				END_CASE
			MS_Running :
				IF (NOT sCurrentState.bWaitStep) THEN
(*----------------- Probing ------------------*)
					FOR iSide := 0 TO 1 DO
						CASE aeProbingStep[iSide] OF
							SP_RunStp1 :
								IF abDoProbing[iSide] THEN
									aiProbingCount[iSide] := 0;
									alrProbingStartPos[iSide] := alrTargetPos[PA_Z1 + iSide];
									abProbingDone[iSide] := FALSE;
									abStartPearlingMotor[iSide] := FALSE;
									aeProbingStep[iSide] := SP_RunStp20;
								END_IF
							SP_RunStp20:
								(* Continuous move probing with analog sensor *)
								IF (aTRobotAxis[PA_Z1+ iSide].eCurrentState = AS_InPosition) AND aTWaitMotorStopped[iSide].Q THEN
									(* Move 0.5 mm above probing pos to check default sensor value *)
									alrTargetPos[PA_Z1 + iSide] := alrProbingStartPos[iSide] - 0.5;		// TODO : HFO modifier valeur en dure, original 0.5
									alrCurrentSpeed[PA_Z1 + iSide] := alrMaxRobotSpeed[PA_Z1 + iSide];
									aeMoveRobotCommand[PA_Z1 + iSide] := AC_MoveAtAbsPos;
									aTStickContactValidated[iSide](IN := FALSE);
									aeProbingStep[iSide] := SP_RunStp21;
								END_IF
							SP_RunStp21:
								IF (aTRobotAxis[PA_Z1 + iSide].eCurrentState = AS_InPosition) THEN
									aTStickContactValidated[iSide](IN := TRUE,PT := TStickStabilisationTime);	// Valueur original ==> PT := TStickContactValidTime
									IF aTStickContactValidated[iSide].Q THEN
										asProbingLog[iSide].iPreviousProbingThreshold := aiContactThresholdArea[iSide , aeProbingArea[iSide]];
										aiContactThresholdArea[iSide , aeProbingArea[iSide]] := aiContactDistance[iSide];
										(* Move down 0.5mm *)
										alrTargetPos[PA_Z1 + iSide] := alrProbingStartPos[iSide]- 0.3;  		// TODO : HFO, Ajout de valeur negative
										//alrTargetPos[PA_Z1 + iSide] := alrProbingStartPos[iSide];
										aeMoveRobotCommand[PA_Z1 + iSide] := AC_MoveAtAbsPos;
										aTStickContactValidated[iSide](IN := FALSE);
										aeProbingStep[iSide] := SP_RunStp25;
									END_IF
								END_IF
							SP_RunStp25:
								IF (aTRobotAxis[PA_Z1 + iSide].eCurrentState = AS_InPosition) THEN
									aTStickContactValidated[iSide](IN := TRUE,PT := TStickContactValidTime);
									IF aTStickContactValidated[iSide].Q THEN
										(* Check if we must go up or down *)
										IF (aiContactDistance[iSide] > aiContactThresholdArea[iSide , aeProbingArea[iSide]] + alrSensorRate[iSide] * lrProbingThreshold) THEN
											(* Go up *)
											aeProbingStep[iSide] := SP_RunStp30;
										ELSE
											(* Go down *)
											aeProbingStep[iSide] := SP_RunStp40;
										END_IF								
									END_IF
								END_IF	
							SP_RunStp30:
								(* Move up slowly until we get contact *)
								alrTargetPos[PA_Z1 + iSide] := alrProbingStartPos[iSide] - 2;
								alrCurrentSpeed[PA_Z1 + iSide] := lrSensorZSpeed;
								aeMoveRobotCommand[PA_Z1 + iSide] := AC_MoveAtAbsPos;
								aeProbingStep[iSide] := SP_RunStp35;
							SP_RunStp35:
								IF (aiContactDistance[iSide] < aiContactThresholdArea[iSide , aeProbingArea[iSide]] + alrSensorRate[iSide] * lrProbingThreshold) THEN
									aTStickContactValidated[iSide](IN := FALSE);
									aeMoveRobotCommand[PA_Z1 + iSide] := AC_Stop;
									aeProbingStep[iSide] := SP_RunStp50;
									sCurrentState.bWaitStep := TRUE;
								ELSIF (aTRobotAxis[PA_Z1 + iSide].eCurrentState = AS_InPosition) THEN
									aeMoveRobotCommand[PA_Z1] := AC_Stop;
									aeMoveRobotCommand[PA_Z2] := AC_Stop;
									bSecurityError := TRUE;
									iDebugPos := 1;
									iDebugSide := iSide;
								END_IF
							SP_RunStp40:
								(* Move down slowly until we get contact *)
								alrTargetPos[PA_Z1 + iSide] := alrProbingLimit[iSide];
								alrCurrentSpeed[PA_Z1 + iSide] := lrSensorZSpeed;
								aeMoveRobotCommand[PA_Z1 + iSide] := AC_MoveAtAbsPos;
								aeProbingStep[iSide] := SP_RunStp45;
							SP_RunStp45:
								IF (aiContactDistance[iSide] > aiContactThresholdArea[iSide , aeProbingArea[iSide]] + alrSensorRate[iSide] * lrProbingThreshold) THEN
									aTStickContactValidated[iSide](IN := FALSE);
									aeMoveRobotCommand[PA_Z1 + iSide] := AC_Stop;
									aeProbingStep[iSide] := SP_RunStp50;
									sCurrentState.bWaitStep := TRUE;
								ELSIF (aTRobotAxis[PA_Z1 + iSide].eCurrentState = AS_InPosition) THEN
									aeMoveRobotCommand[PA_Z1] := AC_Stop;
									aeMoveRobotCommand[PA_Z2] := AC_Stop;
									bSecurityError := TRUE;
									iDebugPos := 10;
									iDebugSide := iSide;
								END_IF
							SP_RunStp50:
								IF (aTRobotAxis[PA_Z1 + iSide].eCurrentState = AS_InPosition) THEN
									aTStickContactValidated[iSide](IN := TRUE,PT := TStickContactValidTime);
									IF aTStickContactValidated[iSide].Q THEN
										alrProbingPos[iSide] := aTRobotAxis[PA_Z1 + iSide].lrCurrentPos - (aiContactDistance[iSide] - aiContactThresholdArea[iSide , aeProbingArea[iSide]])/alrSensorRate[iSide];
										(* Move 2 mm above probing pos to check 1st measure *)
										alrTargetPos[PA_Z1 + iSide] := aTRobotAxis[PA_Z1 + iSide].lrCurrentPos - 2;
										alrCurrentSpeed[PA_Z1 + iSide] := alrMaxRobotSpeed[PA_Z1 + iSide];
										aeMoveRobotCommand[PA_Z1 + iSide] := AC_MoveAtAbsPos;
										aeProbingStep[iSide] := SP_RunStp55;
									END_IF
								END_IF
							SP_RunStp55:
								IF (aTRobotAxis[PA_Z1 + iSide].eCurrentState = AS_InPosition) AND NOT asProbingLog[iSide].bNewLog THEN
									(* Move to contact position *)
									alrTargetPos[PA_Z1 + iSide] := alrTargetPos[PA_Z1 + iSide]+2;
									aeMoveRobotCommand[PA_Z1 + iSide] := AC_MoveAtAbsPos;
									aTStickContactValidated[iSide](IN := FALSE);
									aeProbingStep[iSide] := SP_RunStp60;
								END_IF
							SP_RunStp60:
								IF (aTRobotAxis[PA_Z1 + iSide].eCurrentState = AS_InPosition) THEN
									aTStickContactValidated[iSide](IN := TRUE,PT := TStickContactValidTime);
									IF aTStickContactValidated[iSide].Q THEN
										alrCheckProbingPos[iSide] := aTRobotAxis[PA_Z1 + iSide].lrCurrentPos - (aiContactDistance[iSide] - aiContactThresholdArea[iSide , aeProbingArea[iSide]])/alrSensorRate[iSide];
										asProbingLog[iSide].alrProbingPos[PH_Left] := alrProbingPos[iSide];
										asProbingLog[iSide].alrProbingPos[PH_Right] := alrCheckProbingPos[iSide];
										asProbingLog[iSide].eProbingArea := aeProbingArea[iSide];
										asProbingLog[iSide].iProbingThreshold := aiContactThresholdArea[iSide , aeProbingArea[iSide]];
										asProbingLog[iSide].bNewLog := TRUE;
(* DLA										IF (ABS(alrProbingPos[iSide] - alrCheckProbingPos[iSide]) < 0.1) THEN *)
										IF (ABS(alrProbingPos[iSide] - alrCheckProbingPos[iSide]) < 0.3) THEN
											abProbingDone[iSide] := TRUE;
											aeProbingStep[iSide] := SP_RunStp70;
										ELSIF abRetryProbing[iSide] AND aiProbingCount[iSide] < 3 AND (ABS(alrProbingPos[iSide] - alrCheckProbingPos[iSide]) < 0.3)THEN
											aiProbingCount[iSide] := aiProbingCount[iSide] + 1;
											aeProbingStep[iSide] := SP_RunStp20;
										ELSE
											bSecurityError := TRUE;
											iDebugPos := 2;
											iDebugSide := iSide;
										END_IF
									END_IF
								END_IF
							SP_RunStp70:
								IF NOT abDoProbing[iSide] THEN
									aeProbingStep[iSide] := SP_RunStp1;
								END_IF
						END_CASE
					END_FOR
(*----------------- Stick gestion ------------------*)
					CASE eStickStep OF
						SP_RunStp1 :
							IF (aTRobotAxis[PA_Z1].eCurrentState = AS_InPosition) AND (aTRobotAxis[PA_Z2].eCurrentState = AS_InPosition) THEN
								FOR iSide := 0 TO 1 DO
									IF abChangeStick[iSide] AND abUseSpindle[iSide] THEN
										abSharpenStick[iSide] := TRUE;
										eStickStep := SP_RunStp2; (* Change Stick [Serial]*)
									END_IF
								END_FOR
								IF (eStickStep <> SP_RunStp2) THEN
									FOR iSide := 0 TO 1 DO
										IF abSharpenStick[iSide] AND abUseSpindle[iSide] THEN
											IF NOT abChuckClosed[iSide] THEN
												abSharpenStick[iSide] := FALSE;
											ELSE
												IF abNewStick[iSide] OR aiNbOfPearlsDone[iSide]>0 THEN
													eStickStep := SP_RunStp50; (* Sharpen [parallel]*)
												ELSIF NOT abNewStick[iSide] AND abSharpenStick[iSide] AND aiNbOfPearlsDone[iSide]=0 THEN
													(* sharpen is not need if no pearl has been made *)
													abSharpenStick[iSide] := FALSE;
												END_IF
											END_IF
										END_IF
									END_FOR
								END_IF
							END_IF
						SP_RunStp2 : (* Change Stick [Serial]*)
							FOR iSide := 0 TO 1 DO
								(* Stop motors *)
								abStartPearlingMotor[iSide] := FALSE;
								(* Move Z to safe *)
								alrTargetPos[PA_Z1+iSide] := alrSafePos[PA_Z1+iSide];
								aeMoveRobotCommand[PA_Z1+iSide] := AC_MoveAtAbsPos;
							END_FOR
							eStickStep := SP_RunStp10;
						SP_RunStp10 :  (* Reject Stick [Serial]*)
							IF (aTRobotAxis[PA_Z1].eCurrentState = AS_InPosition) AND
									(aTRobotAxis[PA_Z2].eCurrentState = AS_InPosition) THEN
								eStickStep := SP_RunStp20; (* Nothing to reject, Get new Stick *)
								FOR iSide := 0 TO 1 DO
									(* First drop stick if any *)
									IF abChuckClosed[iSide] AND abChangeStick[iSide] AND abUseSpindle[iSide] THEN
										iRejectPos := iSide;
										eStickStep := SP_RunStp11; (* First drop stick if any *)
										EXIT;
									END_IF
								END_FOR
							END_IF
						SP_RunStp11 :
							(* Move to reject *)
							alrTargetPos[PA_X] := alrRobotPos[PA_X,PTP_RejectPosZ1+iRejectPos];
							alrTargetPos[PA_Y] := alrRobotPos[PA_Y,PTP_RejectPosZ1+iRejectPos];
							aeMoveRobotCommand[PA_X] := AC_MoveAtAbsPos;
							aeMoveRobotCommand[PA_Y] := AC_MoveAtAbsPos;
							eStickStep := SP_RunStp12;
						SP_RunStp12 :
							IF (eRobotXYStatus = AS_InPosition) THEN
								(* Move Z to reject pos *)
								alrTargetPos[PA_Z1+iRejectPos] := alrRobotPos[PA_Z1 + iRejectPos,PTP_RejectPosZ1+iRejectPos];
								aeMoveRobotCommand[PA_Z1+iRejectPos] := AC_MoveAtAbsPos;
								eStickStep := SP_RunStp13;
							END_IF
						SP_RunStp13 :
							IF (aTRobotAxis[PA_Z1+iRejectPos].eCurrentState = AS_InPosition) THEN
								(* Open chuck *)
								abOpenChuck[iRejectPos] := TRUE;
								TCheckTimer(IN := FALSE);
								eStickStep := SP_RunStp14;
							END_IF
						SP_RunStp14 :
							IF abChuckOpened[iRejectPos] THEN
								abActivateEject[iRejectPos] := TRUE;
								TCheckTimer(IN := TRUE,PT := TCheckTime);
								IF TCheckTimer.Q THEN
									abActivateEject[iRejectPos] := FALSE;
									alrTargetPos[PA_Z1+iRejectPos] := alrSafePos[PA_Z1+iRejectPos];
									aeMoveRobotCommand[PA_Z1+iRejectPos] := AC_MoveAtAbsPos;
									eStickStep :=  SP_RunStp10;
								END_IF
							ELSE
								TCheckTimer(IN := FALSE);
							END_IF
						SP_RunStp20 :  (* Get new stick [Serial]*)
							IF (aTRobotAxis[PA_Z1].eCurrentState = AS_InPosition) AND
									(aTRobotAxis[PA_Z2].eCurrentState = AS_InPosition) THEN
								eStickStep := SP_RunStp1; (* Nothing to change *)
								FOR iSide := 0 TO 1 DO
									IF abChangeStick[iSide]  AND abUseSpindle[iSide] THEN
										iChangeStickPos := iSide;
										eStickStep := SP_RunStp21; (* Get new stick *)
										EXIT;
									END_IF
								END_FOR
							END_IF
						SP_RunStp21 :
							iStickHead := iChangeStickPos+1;
							eBarrelRunCmd := RCB_PrepareStick;
							alrTargetPos[PA_X] := alrRobotPos[PA_X,PTP_BarrelPosZ1+iChangeStickPos];
							alrTargetPos[PA_Y] := alrRobotPos[PA_Y,PTP_BarrelPosZ1+iChangeStickPos];
							aeMoveRobotCommand[PA_X] := AC_MoveAtAbsPos;
							aeMoveRobotCommand[PA_Y] := AC_MoveAtAbsPos;
							eStickStep := SP_RunStp22;
						SP_RunStp22 :
							IF (eRobotXYStatus = AS_InPosition) AND (eBarrelRunStatus= RS_WaitRequest ) THEN
								sOutTakeFromBarrel.bHasTaken := FALSE;
								sOutTakeFromBarrel.bReadyToTake := FALSE;
								eBarrelRunCmd := RCB_GiveStick;
								eStickStep := SP_RunStp23;
							END_IF
						SP_RunStp23 :
							IF (eRobotXYStatus = AS_InPosition)  THEN
								(* Move Z to stick pos *)
								alrTargetPos[PA_Z1+iChangeStickPos] := alrRobotPos[PA_Z1+iChangeStickPos,PTP_BarrelPosZ1+iChangeStickPos];
								aeMoveRobotCommand[PA_Z1+iChangeStickPos] := AC_MoveAtAbsPos;
								eStickStep := SP_RunStp24;
							END_IF
						SP_RunStp24 :
							IF (ABS(aTRobotAxis[PA_Z1+iChangeStickPos].lrCurrentPos - alrTargetPos[PA_Z1+iChangeStickPos]) <= 10) THEN
								(* reduce speed when take stick *)
								alrCurrentSpeed[PA_Z1+iChangeStickPos] := lrStickTakeSpeed;
							END_IF
							IF (aTRobotAxis[PA_Z1+iChangeStickPos].eCurrentState = AS_InPosition) THEN
								alrCurrentSpeed := alrMaxRobotSpeed;
								sOutTakeFromBarrel.bReadyToTake := TRUE;
								eStickStep := SP_RunStp25;
							END_IF
						SP_RunStp25 :
							IF sInTakeFromBarrel.bHasGiven THEN
								(* Close chuck *)
								abOpenChuck[iChangeStickPos] := FALSE;
								eStickStep := SP_RunStp26;
							END_IF
						SP_RunStp26 :
							IF abChuckClosed[iChangeStickPos] THEN
								abNewStick[iChangeStickPos] := TRUE;
								(* Move Z to safe *)
								alrTargetPos[PA_Z1+iChangeStickPos] := alrSafePos[PA_Z1+iChangeStickPos];
								aeMoveRobotCommand[PA_Z1+iChangeStickPos] := AC_MoveAtAbsPos;
								eStickStep := SP_RunStp27;
							END_IF
						SP_RunStp27 :
							IF (aTRobotAxis[PA_Z1+iChangeStickPos].eCurrentState = AS_InPosition) THEN
								sOutTakeFromBarrel.bHasTaken := TRUE;
								eStickStep := SP_RunStp28;
							END_IF
						SP_RunStp28 :
							IF eBarrelRunStatus = RS_WaitRequest  THEN
								IF sInTakeFromBarrel.bHasGiven THEN
									abChangeStick[iChangeStickPos] := FALSE;
									abSharpenStick[iChangeStickPos] := TRUE;
									alrRemainingStickLength[iChangeStickPos] := asStickData[iChangeStickPos].lrTotalLength;
									eStickStep := SP_RunStp20;
								ELSE
									bStickNotTakenError := TRUE;
									abSpindleError[iChangeStickPos] := TRUE;
									abOpenChuck[iChangeStickPos] := TRUE;
									eStickStep := SP_RunStp1;  (*Error *)
								END_IF
							END_IF
						SP_RunStp50 : (* Sharpen [parallel]*)
							IF (eSharpenRunStatus =  RS_WaitRequest) THEN
								FOR iSide := 0 TO 1 DO
									(* Stop motors *)
									abStartPearlingMotor[iSide] := FALSE;
									(* Move Z to safe *)
									alrTargetPos[PA_Z1+iSide] := alrSafePos[PA_Z1+iSide];
									aeMoveRobotCommand[PA_Z1+iSide] := AC_MoveAtAbsPos;
								END_FOR
								eStickStep := SP_RunStp51;
							END_IF
						SP_RunStp51 :
							IF (aTRobotAxis[PA_Z1].eCurrentState = AS_InPosition) AND
									(aTRobotAxis[PA_Z2].eCurrentState = AS_InPosition) THEN
								alrTargetPos[PA_X] := alrRobotPos[PA_X,PTP_Sharpen];
								alrTargetPos[PA_Y] := alrRobotPos[PA_Y,PTP_Sharpen];
								aeMoveRobotCommand[PA_X] := AC_MoveAtAbsPos;
								aeMoveRobotCommand[PA_Y] := AC_MoveAtAbsPos;
								eStickStep := SP_RunStp52;
							END_IF
						SP_RunStp52 :
							IF (eRobotXYStatus = AS_InPosition)  THEN
								(* Move Z to sharpen pos if needed*)
								FOR iSide := 0 TO 1 DO
									IF abSharpenStick[iSide]  AND abUseSpindle[iSide] THEN
										(* After sharpening, pearling correction must be recalculated *)
										alrCorrectionMCR[iSide] := 0;
										IF abNewStick[iSide] THEN
											alrTargetPos[PA_Z1+iSide] := alrRobotPos[PA_Z1+iSide,PTP_Sharpen] - lrStickOutAfterChange - 0.5;
										ELSE
											alrTargetPos[PA_Z1+iSide] := alrRobotPos[PA_Z1+iSide,PTP_Sharpen] - lrSharpenPosOffset - asStickData[iSide].lrOutLength;
										END_IF
										aeMoveRobotCommand[PA_Z1+iSide] := AC_MoveAtAbsPos;
									END_IF
								END_FOR
								alrCurrentSpeed := alrMaxRobotSpeed;
								eStickStep := SP_RunStp53;
							END_IF
						SP_RunStp53 :
							IF (aTRobotAxis[PA_Z1].eCurrentState = AS_InPosition) AND
									(aTRobotAxis[PA_Z2].eCurrentState = AS_InPosition) THEN
								FOR iSide := 0 TO 1 DO
									IF abSharpenStick[iSide]  AND abUseSpindle[iSide] THEN
										IF NOT abNewStick[iSide] THEN
											alrProbingLimit[iSide] :=  alrRobotPos[PA_Z1+iSide,PTP_Sharpen] + 0.5;
											abDoProbing[iSide] := TRUE;
											abRetryProbing[iSide] := FALSE;
										END_IF
										aeProbingArea[iSide] := PA_BeforeSharpen;
									END_IF
								END_FOR
								eStickStep := SP_RunStp54;
							END_IF
						SP_RunStp54 :
							IF (abProbingDone[PH_Left] OR NOT abSharpenStick[PH_Left] OR NOT abUseSpindle[PH_Left] OR abNewStick[PH_Left]) AND (abProbingDone[PH_Right] OR NOT abSharpenStick[PH_Right] OR  NOT abUseSpindle[PH_Right] OR abNewStick[PH_Right]) THEN
								FOR iSide := 0 TO 1 DO
									abDoProbing[iSide] := FALSE;
									(* We have the right position, calculate stick use *)
									IF abSharpenStick[iSide]   AND abUseSpindle[iSide] THEN
										IF abNewStick[iSide] THEN
											alrRemainingStickLength[iSide] := asStickData[iSide].lrTotalLength;
										ELSE
											IF (alrProbingPos[iSide] - alrLastProbingPos[iSide]) > (asStickData[iSide].lrOutLength -0.5) THEN
												alrRemainingStickLength[iSide] := sStickDataShared.sStickDataMMIShared.lrMinHoldLength;
											ELSE
												alrRemainingStickLength[iSide] := alrRemainingStickLength[iSide] - (alrProbingPos[iSide] - alrLastProbingPos[iSide]);
											END_IF
										END_IF
										(* Check if it is the first probing after stick change *)
										IF (alrRemainingStickLength[iSide] > asStickData[iSide].lrTotalLength) THEN
											alrRemainingStickLength[iSide] := asStickData[iSide].lrTotalLength;
										END_IF
										(* Check if the stick is not too short *)
										IF (alrRemainingStickLength[iSide] < (sStickDataShared.sStickDataMMIShared.lrMinHoldLength + asStickData[iSide].lrOutLength)) THEN
											(* We must change the stick *)
											abChangeStick[iSide] := TRUE;
											abSharpenStick[iSide] := FALSE;
											eStickStep := SP_RunStp1;
										END_IF
									END_IF
								END_FOR
								IF (eStickStep = SP_RunStp1) THEN
									(* In parallel pearling, we must change both stick *)
									IF bParallelProduction THEN
										FOR iSide:=0 TO 1 DO
											abChangeStick[iSide] := TRUE;
											abSharpenStick[iSide] := FALSE;
										END_FOR
									END_IF
								ELSE
									FOR iSide := 0 TO 1 DO
										IF abSharpenStick[iSide]   AND abUseSpindle[iSide] AND NOT abNewStick[iSide] THEN
											alrTargetPos[PA_Z1+iSide] := alrTargetPos[PA_Z1+iSide] - 0.5;
											aeMoveRobotCommand[PA_Z1+iSide] := AC_MoveAtAbsPos;
										END_IF
									END_FOR
									eStickStep := SP_RunStp55;
								END_IF
							END_IF
						SP_RunStp55 :
							IF (aTRobotAxis[PA_Z1].eCurrentState = AS_InPosition) AND
								(aTRobotAxis[PA_Z2].eCurrentState = AS_InPosition) THEN
								FOR iSide := 0 TO 1 DO
									IF   abUseSpindle[iSide] AND abSharpenStick[iSide] THEN
										(* Open chuck *)
										abOpenChuck[iSide] := TRUE;
									END_IF
								END_FOR
								TWaitChuckOpen(IN := FALSE);
								eStickStep := SP_RunStp56;
							END_IF
						SP_RunStp56 :
							TWaitChuckOpen(IN := (abChuckOpened[PH_Left] OR NOT abOpenChuck[PH_Left] OR NOT abUseSpindle[PH_Left]) AND (abChuckOpened[PH_Right] OR NOT abOpenChuck[PH_Right] OR NOT abUseSpindle[PH_Right]),PT := T#400MS);   // Valeur de départ ==> PT := t#1s
							FOR iSide := 0 TO 1 DO
								IF abUseSpindle[iSide] AND abSharpenStick[iSide] THEN
									abActivateEject[iSide] := abChuckOpened[iSide] AND abOpenChuck[iSide];
									IF  TWaitChuckOpen.Q THEN
										(* Move Z to out position *)
										alrCurrentSpeed := alrMaxRobotSpeed;
										alrTargetPos[PA_Z1+iSide] := alrRobotPos[PA_Z1+iSide,PTP_Sharpen]- asStickData[iSide].lrOutLength - alrSharpenTeachZOffset;
										aeMoveRobotCommand[PA_Z1+iSide] := AC_MoveAtAbsPos;
										//eStickStep := SP_RunStp57;		// HFO : Supprimer la correction avec capteur step 57, 58, 24.11.2021
										eStickStep := SP_RunStp59;
									END_IF
								END_IF
							END_FOR
						SP_RunStp57:
							IF (aTRobotAxis[PA_Z1].eCurrentState = AS_InPosition) AND
								(aTRobotAxis[PA_Z2].eCurrentState = AS_InPosition) THEN
								TWaitHeadStab(IN := FALSE);
								eStickStep := SP_RunStp58;
							END_IF
						SP_RunStp58:
							TWaitHeadStab(IN := TRUE, PT := T#150MS);	// Valeur de départ ==> PT := t#500ms
							IF TWaitHeadStab.Q THEN
								FOR iSide := 0 TO 1 DO
									IF abUseSpindle[iSide] AND abSharpenStick[iSide] THEN
										alrTargetPos[PA_Z1+iSide] := alrTargetPos[PA_Z1+iSide] + (aiContactDistance[iSide] - aiContactThresholdArea[iSide , aeProbingArea[iSide]])/alrSensorRate[iSide] - alrChuckRetractOffset[iSide];
										aeMoveRobotCommand[PA_Z1+iSide] := AC_MoveAtAbsPos;
									END_IF
								END_FOR
								eStickStep := SP_RunStp59;
							END_IF
						SP_RunStp59:
							IF (aTRobotAxis[PA_Z1].eCurrentState = AS_InPosition) AND
									(aTRobotAxis[PA_Z2].eCurrentState = AS_InPosition) THEN
								TWaitHeadStab(IN := FALSE);
								eStickStep := SP_RunStp60;
							END_IF
						SP_RunStp60:
							TWaitHeadStab(IN := TRUE, PT := T#400MS);	// Valeur de départ ==> PT := t#500ms
							IF TWaitHeadStab.Q THEN
								eStickStep := SP_RunStp61;
							END_IF
						SP_RunStp61 :
							IF (aTRobotAxis[PA_Z1].eCurrentState = AS_InPosition) AND
									(aTRobotAxis[PA_Z2].eCurrentState = AS_InPosition) THEN
								(* Close chuck if needed*)
								FOR iSide := 0 TO 1 DO
									IF abUseSpindle[iSide] AND abSharpenStick[iSide] THEN
										abOpenChuck[iSide] := FALSE;
									END_IF
								END_FOR
								IF (abChuckClosed[PH_Left]  OR abOpenChuck[PH_Left] OR NOT abUseSpindle[PH_Left]) AND (abChuckClosed[PH_Right] OR abOpenChuck[PH_Right] OR NOT abUseSpindle[PH_Right]) THEN
									FOR iSide := 0 TO 1 DO
										IF abUseSpindle[iSide] AND abSharpenStick[iSide] THEN
											(* Retract ejector *)
											abActivateEject[iSide] := FALSE;
											(* Do probing *)
											alrTargetPos[PA_Z1+iSide] := alrTargetPos[PA_Z1+iSide];
(* DLA : Remove -1mm for optimisation 											alrTargetPos[PA_Z1+iSide] := alrTargetPos[PA_Z1+iSide] - 1;*)
											alrProbingLimit[iSide] :=  alrRobotPos[PA_Z1+iSide,PTP_Sharpen] - 0.5;
											abDoProbing[iSide] := TRUE;
											abRetryProbing[iSide] := FALSE;
											aeProbingArea[iSide] := PA_AfterSharpen;
										END_IF
									END_FOR
									eStickStep := SP_RunStp62;
								END_IF
							END_IF
						SP_RunStp62 :
							IF (abProbingDone[PH_Left] OR NOT abSharpenStick[PH_Left]  OR NOT abUseSpindle[PH_Left]) AND (abProbingDone[PH_Right] OR NOT abSharpenStick[PH_Right] OR NOT abUseSpindle[PH_Right]) THEN
								alrCurrentSpeed := alrMaxRobotSpeed;
								FOR iSide := 0 TO 1 DO
									IF abUseSpindle[iSide] AND abSharpenStick[iSide] THEN
										alrLastProbingPos[iSide] := alrProbingPos[iSide];
										alrSharpenProbing[iSide] := alrProbingPos[iSide];
										alrStickCorrection[iSide] := alrRobotPos[PA_Z1+iSide,PTP_Sharpen]  - alrProbingPos[iSide] - asStickData[iSide].lrOutLength - alrSharpenTeachZOffset;
										(* Move down to sharpen end position*)
										alrTargetPos[PA_Z1+iSide] := alrProbingPos[iSide] - 0.1;
										aeMoveRobotCommand[PA_Z1+iSide] := AC_MoveAtAbsPos;
										(* Check if there is a risk for the spindle or stick is stuck in the chuck*)
										IF (alrProbingPos[iSide] > ( alrRobotPos[PA_Z1+iSide,PTP_Sharpen] - (asStickData[iSide].lrOutLength - 0.5))) THEN
											abChangeStick[iSide] := TRUE;
											bSecurityError := TRUE;
											iDebugPos := 3;
											iDebugSide := iSide;
										END_IF
									END_IF
								END_FOR
								IF bSecurityError THEN
									aeMoveRobotCommand[PA_Z1] := AC_None;
									aeMoveRobotCommand[PA_Z2] := AC_None;
								ELSE
									bAspirationSharpenOn := TRUE;
									eStickStep := SP_RunStp63;
								END_IF
							END_IF
						SP_RunStp63 :
							IF (aTRobotAxis[PA_Z1].eCurrentState = AS_InPosition) AND
									(aTRobotAxis[PA_Z2].eCurrentState = AS_InPosition) THEN
								IF bUseFullTapeWidth THEN
									(* Move to start position *)
									alrCurrentSpeed := alrMaxRobotSpeed;
									alrTargetPos[PA_Y] := alrRobotPos[PA_Y,PTP_Sharpen] - lrCenterSharpningOffset - lrSharpeningDelta;
									aeMoveRobotCommand[PA_Y] := AC_MoveAtAbsPos;
								END_IF
								yMCRChannel := 1;
								eStickStep := SP_RunStp64;
							END_IF
						SP_RunStp64 :
							eMCRCommand := MCRC_SetSpeed;
							TMCRDrv.iSpeedSetpoint :=  sStickDataShared.sStickDataMMIShared.iMCRSharpenSpeed;
							eStickStep := SP_RunStp65;
						SP_RunStp65 :
							IF bMCRReady THEN
								IF yMCRChannel = 1 THEN
									yMCRChannel := 2;
									eStickStep := SP_RunStp64;
								ELSE
									yMCRChannel := 1;
									eStickStep := SP_RunStp66;
								END_IF
							END_IF
						SP_RunStp66:
							(* Wait XY in start position *)
							IF (eRobotXYStatus = AS_InPosition) THEN
								FOR iSide := 0 TO 1 DO
									IF abUseSpindle[iSide] AND abSharpenStick[iSide] THEN
										abStartPearlingMotor[iSide] := TRUE;
									END_IF
								END_FOR
								IF  (aTWaitMotorStarted[PH_Left].Q OR NOT abSharpenStick[PH_Left] OR NOT abUseSpindle[PH_Left]) AND (aTWaitMotorStarted[PH_Right].Q OR NOT abSharpenStick[PH_Right] OR NOT abUseSpindle[PH_Right])   THEN
									FOR iSide := 0 TO 1 DO
										IF abUseSpindle[iSide] AND abSharpenStick[iSide] THEN
											abDoProbing[iSide] := FALSE;
											(* Move down to sharpen end position*)
											IF abNewStick[iSide] THEN
												alrTargetPos[PA_Z1+iSide] := alrTargetPos[PA_Z1+iSide] + 0.2 +0.05;
											ELSE
												alrTargetPos[PA_Z1+iSide] := alrTargetPos[PA_Z1+iSide] + sStickDataShared.sStickDataMMIShared.lrSharpenHeight+0.05;
											END_IF
											aeMoveRobotCommand[PA_Z1+iSide] := AC_MoveAtAbsPos;
											abNewStick[iSide] := FALSE;
										END_IF
									END_FOR
									alrCurrentSpeed := alrMaxRobotSpeed;
									iNbOfFwBwSharpen := 0;
									iNbOfFwBwSharpenBeforeMove := 0;
									eStickStep := SP_RunStp67;
								END_IF
							END_IF
						SP_RunStp67 :
							IF  (aTRobotAxis[PA_Z1].eCurrentState = AS_InPosition) AND (aTRobotAxis[PA_Z2].eCurrentState = AS_InPosition) THEN
								(* Reduce speed for sharpening *)
								alrCurrentSpeed[PA_Y] := sStickDataShared.sStickDataMMIShared.lrSharpenSpeed;
								eStickStep := SP_RunStp68;
							END_IF
						SP_RunStp68 :
							(* Do sharpening *)
							IF (eRobotXYStatus = AS_InPosition) THEN
								iNbOfFwBwSharpen := iNbOfFwBwSharpen+1;
								iNbOfFwBwSharpenBeforeMove := iNbOfFwBwSharpenBeforeMove + 1;
								(* Check if sharpen is finished *)
								IF (iNbOfFwBwSharpen >  sStickDataShared.sStickDataMMIShared.iNbOfFwBwSharpen) THEN
									eStickStep := SP_RunStp71;
								ELSE
									eStickStep := SP_RunStp69;
									IF bUseFullTapeWidth THEN
										IF iNbOfFwBwSharpen = 1 THEN
											alrTargetPos[PA_Y] := alrRobotPos[PA_Y,PTP_Sharpen] - lrCenterSharpningOffset - lrSharpeningDelta;
											eStickStep := SP_RunStp80;
										ELSE
											alrTargetPos[PA_Y] := alrRobotPos[PA_Y,PTP_Sharpen] - lrCenterSharpningOffset;
										END_IF
									ELSE
										alrTargetPos[PA_Y] := alrRobotPos[PA_Y,PTP_Sharpen] - lrCenterSharpningOffset + lrSharpeningDelta;
									END_IF
									aeMoveRobotCommand[PA_Y] := AC_MoveAtAbsPos;
								END_IF
							END_IF
						SP_RunStp69 :
							(* Do sharpening *)
							IF (eRobotXYStatus = AS_InPosition) THEN
								eStickStep := SP_RunStp68;
								IF (iNbOfFwBwSharpenBeforeMove >= sStickDataShared.sStickDataMMIShared.iNbOfFwBwBeforeTapeMove) OR
											(iNbOfFwBwSharpen = sStickDataShared.sStickDataMMIShared.iNbOfFwBwSharpen) THEN
									IF bUseFullTapeWidth THEN
										(* Move on clean tape part *)
										alrTargetPos[PA_Y] := alrRobotPos[PA_Y,PTP_Sharpen] - lrCenterSharpningOffset + lrSharpeningDelta;
										aeMoveRobotCommand[PA_Y] := AC_MoveAtAbsPos;
									ELSE
										(* Move Sharpen Tape*)
										eSharpenRunCmd := RCS_MoveStep;
										eStickStep := SP_RunStp70;
									END_IF
									iNbOfFwBwSharpenBeforeMove := 0;
								ELSIF bUseFullTapeWidth THEN
									(* Move BW *)
									alrTargetPos[PA_Y] := alrRobotPos[PA_Y,PTP_Sharpen] - lrCenterSharpningOffset - lrSharpeningDelta;
									aeMoveRobotCommand[PA_Y] := AC_MoveAtAbsPos;
								END_IF
							END_IF
						SP_RunStp70 :
							IF eSharpenRunStatus =  RS_WaitRequest THEN
								alrTargetPos[PA_Y] := alrRobotPos[PA_Y,PTP_Sharpen];
								aeMoveRobotCommand[PA_Y] := AC_MoveAtAbsPos;
								eStickStep := SP_RunStp68;
							END_IF
						SP_RunStp71 :
							(* End of  sharpening *)
							IF (eRobotXYStatus = AS_InPosition) THEN
								IF bUseFullTapeWidth THEN
									(* Move Sharpen Tape*)
									eSharpenRunCmd := RCS_MoveStep;
								END_IF
								(* Take maximal speed *)
								alrCurrentSpeed := alrMaxRobotSpeed;
								(* Move Z to safe *)
								alrTargetPos[PA_Z1] := alrSafePos[PA_Z1];
								alrTargetPos[PA_Z2] := alrSafePos[PA_Z2];
								aeMoveRobotCommand[PA_Z1] := AC_MoveAtAbsPos;
								aeMoveRobotCommand[PA_Z2] := AC_MoveAtAbsPos;
								eStickStep := SP_RunStp72;
							END_IF
						SP_RunStp72:
							IF (aTRobotAxis[PA_Z1].eCurrentState = AS_InPosition) AND
									(aTRobotAxis[PA_Z2].eCurrentState = AS_InPosition) THEN
								bAspirationSharpenOn := FALSE;
								yMCRChannel := 1;
								eStickStep := SP_RunStp73;
							END_IF
						SP_RunStp73 :
							eMCRCommand := MCRC_SetSpeed;
							TMCRDrv.iSpeedSetpoint := sRunData.sPearlingData.iMCRSpeed;
							eStickStep := SP_RunStp74;
						SP_RunStp74 :
							IF bMCRReady THEN
								IF yMCRChannel = 1 THEN
									yMCRChannel := 2;
									eStickStep := SP_RunStp73;
								ELSE
									yMCRChannel := 1;
									eStickStep := SP_RunStp76;
								END_IF
							END_IF
						SP_RunStp76:
							IF  (aTWaitMotorStarted[PH_Left].Q OR NOT abSharpenStick[PH_Left] OR NOT abUseSpindle[PH_Left]) AND (aTWaitMotorStarted[PH_Right].Q OR NOT abSharpenStick[PH_Right] OR NOT abUseSpindle[PH_Right])   THEN
								FOR iSide := 0 TO 1 DO
									IF abUseSpindle[iSide] AND abSharpenStick[iSide] THEN
										aiNbOfPearlsDone[iSide] := 0;
										abSharpenStick[iSide] := FALSE;
									END_IF
								END_FOR
								eStickStep := SP_RunStp1;
							END_IF
						SP_RunStp80 :
							(* Optimised case for using full tape and 1 FwBw *)
							IF (eRobotXYStatus = AS_InPosition) THEN
								alrTargetPos[PA_Y] := alrRobotPos[PA_Y,PTP_Sharpen] - lrCenterSharpningOffset + lrSharpeningDelta;
								aeMoveRobotCommand[PA_Y] := AC_MoveAtAbsPos;
								eStickStep := SP_RunStp68;
							END_IF
					END_CASE
(*----------------- Run ------------------*)
					CASE sCurrentState.eStep OF
						SP_RunStp1 :
							eRunStatus := RS_WaitRequest;
							CASE eRunCommand OF
								RCP_None:
									IF ((NOT abChangeStick[PH_Left] AND NOT abSharpenStick[PH_Left])  OR NOT abUseSpindle[PH_Left]) AND
										((NOT abChangeStick[PH_Right] AND NOT abSharpenStick[PH_Right])  OR NOT abUseSpindle[PH_Right]) THEN
										IF bStopReq  THEN
											sCurrentState.eStatus := MS_Ready;
										ELSIF bPauseReq  THEN
											sCurrentState.eStatus := MS_Paused;
										END_IF
									END_IF
								RCP_Pearl:
									sCurrentState.eStep := SP_RunStp2;
								RCP_CheckSharpen:
									sCurrentState.eStep := SP_RunStp210;
								RCP_ChangeChuck:
									sCurrentState.eStep := SP_RunStp200;
							END_CASE
							IF sCurrentState.eStep<> SP_RunStp1 THEN eRunStatus := RS_ProcessRequest1; END_IF
						SP_RunStp2:(* Pearling startup *)
							(* wait until all sharpening is finish for current used head*)
							IF ((NOT abChangeStick[PH_Left] AND NOT abSharpenStick[PH_Left])  OR NOT abUseSpindle[PH_Left]) AND
								((NOT abChangeStick[PH_Right] AND NOT abSharpenStick[PH_Right])  OR NOT abUseSpindle[PH_Right]) THEN
									alrCurrentSpeed[PA_Z1] := alrMaxRobotSpeed[PA_Z1];
									alrCurrentSpeed[PA_Z2] := alrMaxRobotSpeed[PA_Z2];
									sCurrentState.bWaitStep := TRUE;
									sCurrentState.eStep := SP_RunStp3;
							END_IF
						SP_RunStp3: (* it's now safe to switch head used *)
							abUseSpindle := sRunData.abUseSpindle;
							FOR iSide:=0 TO 1 DO
								IF (NOT abChuckClosed[iSide] OR abNeedChangeStick[iSide]) AND abUseSpindle[iSide] THEN
									abNeedChangeStick[iSide] := FALSE;
									abChangeStick[iSide] := TRUE;
								END_IF
							END_FOR
							sCurrentState.eStep := SP_RunStp4;
						SP_RunStp4 :
							IF ((NOT abChangeStick[PH_Left] AND NOT abSharpenStick[PH_Left])  OR NOT abUseSpindle[PH_Left]) AND
								((NOT abChangeStick[PH_Right] AND NOT abSharpenStick[PH_Right])  OR NOT abUseSpindle[PH_Right]) THEN
									alrCurrentSpeed[PA_Z1] := alrMaxRobotSpeed[PA_Z1];
									alrCurrentSpeed[PA_Z2] := alrMaxRobotSpeed[PA_Z2];
									sCurrentState.eStep := SP_RunStp5;
							END_IF
						SP_RunStp5 :
							IF NOT asPearlData[PH_Left].bNewPart AND NOT asPearlData[PH_Right].bNewPart THEN
								FOR i := 0 TO C_MAX_NB_OF_PEARLS  DO
									aArea[i].iFirstPearl := -1;
									aArea[i].iNbOfPearls := 0;
								END_FOR
								sCurrentState.eStep := SP_RunStp6;
							END_IF
						SP_RunStp6:
							(* Init pearling parameter *)
							FOR i := 1 TO UINT_TO_INT(sRunData.sPearlingData.nNbOfPearls)-1  DO
								IF NOT sRunData.sPearlingData.aDataPerlage[i].bDisable THEN
									iCurrentArea := sRunData.sPearlingData.aDataPerlage[i].iArea;
									aArea[iCurrentArea].iNbOfPearls := aArea[iCurrentArea].iNbOfPearls + 1;
									IF aArea[iCurrentArea].iFirstPearl = -1 THEN aArea[iCurrentArea].iFirstPearl := i; END_IF
								END_IF
							END_FOR
							FOR iSide := 0 TO 1 DO
								anPearlIndexDone[iSide] := 0;
								aiCountPearlError[iSide] := 0;
								abFirstPearl[iSide] := TRUE;
								abNeedChangeStick[iSide] := FALSE;
								aiPearlingLayringPos[iSide] := sRunData.iLayringPos;
								aiPearlingLayringOffsetPos[iSide] := sRunData.iLayringOffsetPos;
								IF abUseSpindle[iSide] THEN
									asPearlData[iSide].bPearlingTop := (sRunData.apsPartData[iSide]^.ePartSide = PS_SUS);
									asPearlData[iSide].bNewPart := TRUE;
									anPearlIndexDone[iSide] := sRunData.apsPartData[iSide]^.anLastPearlIndexDone[aiSideInfo[iSide],sRunData.apsPartData[iSide]^.ePartSide];
								END_IF
							END_FOR
							IF abUseSpindle[PH_Left] THEN
								iFirstHeadUsed := 0;
								IF abUseSpindle[PH_Right] THEN
									aiPearlingLayringPos[PH_Right] := aiPearlingLayringPos[PH_Right] + 1;
								END_IF
							ELSE
								iFirstHeadUsed := 1;
							END_IF
							IF eTableSideForLoader = TS_A THEN (* pearling use the other side *)
								FOR iSide := 0 TO 1 DO
									aiPearlingLayringPos[iSide] := aiPearlingLayringPos[iSide] + 2;
								END_FOR
							END_IF
							nPearlIndex := anPearlIndexDone[PH_Left] + 1;
							IF anPearlIndexDone[PH_Right] + 1 < nPearlIndex THEN nPearlIndex := anPearlIndexDone[PH_Right] + 1; END_IF
							IF nPearlIndex < 1 THEN nPearlIndex := 1; END_IF
							iCurrentArea := -1; (* Force check of sharpening *)
							FOR iSide := 0 TO 1 DO
								IF abUseSpindle[iSide] THEN
									abAspirationPearling[aiPearlingLayringPos[iSide]  MOD 2] := TRUE;
								END_IF
								abTakeZRef[iSide] := NOT abZRefTaken[aiPearlingLayringPos[iSide], aiPearlingLayringOffsetPos[iSide], iSide] AND abUseSpindle[iSide];
								IF bForceProbing THEN
									abTakeZRef[iSide]:= abUseSpindle[iSide];
									abStartPearlingMotor[iSide] := FALSE;
								 END_IF
							END_FOR
							(* First move Z to safe *)
							alrTargetPos[PA_Z1] := alrSafePos[PA_Z1];
							alrTargetPos[PA_Z2] := alrSafePos[PA_Z2];
							aeMoveRobotCommand[PA_Z1] := AC_MoveAtAbsPos;
							aeMoveRobotCommand[PA_Z2] := AC_MoveAtAbsPos;
							sCurrentState.eStep := SP_RunStp7;
						SP_RunStp7:
							IF (aTRobotAxis[PA_Z1].eCurrentState = AS_InPosition) AND
									(aTRobotAxis[PA_Z2].eCurrentState = AS_InPosition) THEN
								IF (aiPearlingLayringPos[iFirstHeadUsed] > 1) THEN (* Handle offset for table Side A/B *)
									aiPearlingTeachedPos[PH_Left] := PTP_TableSideBPosZ1;
									aiPearlingTeachedPos[PH_Right] := PTP_TableSideBPosZ2;
								ELSE
									aiPearlingTeachedPos[PH_Left] := PTP_TableSideAPosZ1;
									aiPearlingTeachedPos[PH_Right] := PTP_TableSideAPosZ2;
								END_IF
								IF abUseSpindle[PH_Left] THEN (* Handle offset for head *)
									alrPearlingOffset[PA_X] := alrRobotPos[PA_X,aiPearlingTeachedPos[PH_Left]];
									alrPearlingOffset[PA_Y] := alrRobotPos[PA_Y,aiPearlingTeachedPos[PH_Left]];
								ELSE
									alrPearlingOffset[PA_X] := alrRobotPos[PA_X,aiPearlingTeachedPos[PH_Right]];
									alrPearlingOffset[PA_Y] := alrRobotPos[PA_Y,aiPearlingTeachedPos[PH_Right]];
								END_IF
								FOR iSide := 0 TO 1 DO
									alrPearlingOffset[PA_Z1+iSide] :=  alrRobotPos[PA_Z1+iSide,aiPearlingTeachedPos[iSide]];
								END_FOR

								IF ((aiPearlingLayringPos[iFirstHeadUsed] MOD 2 )= 0) THEN (* Handle offset for layring*)
									alrPearlingOffset[PA_X] := alrPearlingOffset[PA_X] - lrLayeringCenterOffsetXTable/2;
								ELSE
									alrPearlingOffset[PA_X] := alrPearlingOffset[PA_X] + lrLayeringCenterOffsetXTable/2;
								END_IF
								alrPearlingOffset[PA_Y] := alrPearlingOffset[PA_Y] + lrLayeringCenterOffsetYTable;
								TLayeringCenter.lrX := alrPearlingOffset[PA_X];
								TLayeringCenter.lrY := alrPearlingOffset[PA_Y];
								IF aiPearlingLayringOffsetPos[iFirstHeadUsed] > 0 THEN (* Handle offset for Part on layring*)
									alrPearlingOffset[PA_X] := alrPearlingOffset[PA_X] + sPartData.alrPartOffsetLayering[PH_Right].lrX;
									alrPearlingOffset[PA_Y] := alrPearlingOffset[PA_Y] + sPartData.alrPartOffsetLayering[PH_Right].lrY;
								ELSE
									alrPearlingOffset[PA_X] := alrPearlingOffset[PA_X] + sPartData.alrPartOffsetLayering[PH_Left].lrX;
									alrPearlingOffset[PA_Y] := alrPearlingOffset[PA_Y] + sPartData.alrPartOffsetLayering[PH_Left].lrY;
								END_IF
								(*Check if a pearl is outside of pearling area on layering *)
								FOR nPearl:=0 TO sRunData.sPearlingData.nNbOfPearls - 1 DO
									IF NOT sRunData.sPearlingData.aDataPerlage[nPearl].bDisable THEN
										TPearlPosition.lrX := alrPearlingOffset[PA_X]  + sRunData.sPearlingData.aDataPerlage[nPearl].lrX *alrPearlingInvert[PA_X];
										TPearlPosition.lrY := alrPearlingOffset[PA_Y]  + sRunData.sPearlingData.aDataPerlage[nPearl].lrY *alrPearlingInvert[PA_Y];
										lrRadius := SQRT(EXPT(TPearlPosition.lrX - TLayeringCenter.lrX , 2) + EXPT(TPearlPosition.lrY - TLayeringCenter.lrY, 2));
										IF (lrRadius > lrSecurityRadius) THEN
											bSecurityError := TRUE;
											iDebugPos := 4;
											iDebugSide := -1;
											EXIT;
										END_IF
									END_IF
								END_FOR
								FOR iSide := 0 TO 1 DO
									aePearlingArea[iSide] := PA_PartLayering1Offset0 + aiPearlingLayringPos[iSide] * 2 + aiPearlingLayringOffsetPos[iSide];
								END_FOR
								alrTargetPos[PA_X] := alrPearlingOffset[PA_X];
								alrTargetPos[PA_Y] := alrPearlingOffset[PA_Y];
								aeMoveRobotCommand[PA_X] := AC_MoveAtAbsPos;
								aeMoveRobotCommand[PA_Y] := AC_MoveAtAbsPos ;
								IF abTakeZRef[PH_Left] OR abTakeZRef[PH_Right] THEN
									(* Do referencing on part *)
									sCurrentState.eStep := SP_RunStp30;
								ELSE
									(* Do Pearling *)
									(*abStartPearlingMotor[PH_Left] := TRUE;			// TODO : HFO, problem sometimes when one spindle (spindle 1???) need probing and take ref on part, second spindle don't run
									abStartPearlingMotor[PH_Right] := TRUE;*)
									abUseSpindle[PH_Left] := TRUE;
									abUseSpindle[PH_Right] := TRUE;
									sCurrentState.eStep := SP_RunStp10;
								END_IF
							END_IF
						SP_RunStp10 :
							IF (eRobotXYStatus = AS_InPosition) THEN
								yMCRChannel := 1;
								sCurrentState.eStep := SP_RunStp11;
							END_IF
						SP_RunStp11 :
							(* Do spindle heat on if needed *)
							TMCRDrv.iSpeedSetpoint := iHeatOnSpeed;;
							eMCRCommand := MCRC_SetSpeed;
							sCurrentState.eStep := SP_RunStp12;
						SP_RunStp12 :
							IF bMCRReady THEN
								IF yMCRChannel = 1 THEN
									yMCRChannel := 2;
									sCurrentState.eStep := SP_RunStp11;
								ELSE
									sCurrentState.eStep := SP_RunStp13;
								END_IF
							END_IF
						SP_RunStp13 :
							abStartPearlingMotor[PH_Left] := abNeedSpindleHeatOn[PH_Left];
							abStartPearlingMotor[PH_Right] := abNeedSpindleHeatOn[PH_Right];
							IF (NOT abNeedSpindleHeatOn[PH_Left] AND NOT abNeedSpindleHeatOn[PH_Right]) THEN
								yMCRChannel := 1;
								sCurrentState.eStep := SP_RunStp21;
							END_IF
						SP_RunStp21 :
							eMCRCommand := MCRC_SetSpeed;
							TMCRDrv.iSpeedSetpoint := sRunData.sPearlingData.iMCRSpeed;
							sCurrentState.eStep := SP_RunStp22;
						SP_RunStp22 :
							IF bMCRReady THEN
								IF yMCRChannel = 1 THEN
									yMCRChannel := 2;
									sCurrentState.eStep := SP_RunStp21;
								ELSE
									yMCRChannel := 1;
									sCurrentState.eStep := SP_RunStp23;
								END_IF
							END_IF
						SP_RunStp23 :
							FOR iSide:=0 TO 1 DO
								abSpindleCurrentOk[iSide] := bBypassMCR;
							END_FOR
							TWaitCurrentMotorBeltOk(IN :=FALSE);
							TWaitCurrentMotorWarmOk(IN :=FALSE);
							sCurrentState.eStep := SP_RunStp24;
						SP_RunStp24:
							IF (aTWaitMotorStarted[0].Q OR NOT abUseSpindle[PH_Left]) AND
									(aTWaitMotorStarted[1].Q OR NOT abUseSpindle[PH_Right]) THEN
								IF abSpindleCurrentOk[0] AND abSpindleCurrentOk[1] THEN
									(* Ready to pearl *)
									sCurrentState.eStep := SP_RunStp40;
								ELSE
									(* Pearling can start when current is OK *)
									eMCRCommand := MCRC_GetStatus;
									sCurrentState.eStep := SP_RunStp25;
								END_IF
							END_IF
						SP_RunStp25 : (* Checking spindle current is in range *)
							TWaitCurrentMotorBeltOk(IN :=TRUE,PT := T#5S);
							TWaitCurrentMotorWarmOk(IN :=TRUE,PT := t#10s);
							IF bMCRReady THEN
								// Check status flags
								FOR iSide:=0 TO 1 DO
									IF abUseSpindle[iSide] THEN
										IF TMCRDrv.ayChannelStatus[iSide].1 THEN
											(* Motor belt is ok *)
											IF NOT (TMCRDrv.ayChannelStatus[iSide].3 OR TMCRDrv.ayChannelStatus[iSide].4) THEN
												(* Motor is warm but not over limit *)
												abSpindleCurrentOk[iSide] := TRUE;
											ELSIF TWaitCurrentMotorWarmOk.Q THEN
												IF  TMCRDrv.ayChannelStatus[iSide].4 THEN
													(* Motor is not warm *)
													abCurrentReadError[iSide] := TRUE;
													iDebugSide := iSide;
													IDebugPos := 1;
												ELSE
													(* Motor is warm but over limit*)
													abSpindleCurrentOk[iSide] := TRUE;
													abCurrentLimitWarning[iSide] := TRUE;
													iDebugSide := iSide;
													IDebugPos := 2;
												END_IF
											END_IF
										ELSIF TWaitCurrentMotorBeltOk.Q THEN
											(* Motor belt is not ok *)
											abCurrentReadError[iSide] := TRUE;
										END_IF
									END_IF
								END_FOR
								(* Read current again *)
								sCurrentState.eStep := SP_RunStp24;
							END_IF
						SP_RunStp30:
							IF (aTRobotAxis[PA_Z1].eCurrentState = AS_InPosition) AND
									(aTRobotAxis[PA_Z2].eCurrentState = AS_InPosition) THEN
								FOR iSide := 0 TO 1 DO
									IF sRunData.sPearlingData.iSharpenFreq = 0 AND aiNbOfPearlsDone[iSide] > 0  AND abTakeZRef[iSide] THEN
										(* sharpen is needed before taking ref on part *)
										abSharpenStick[iSide] := TRUE;
									END_IF
								END_FOR
								sCurrentState.eStep := SP_RunStp31;
							END_IF
						SP_RunStp31:
							IF ((NOT abChangeStick[PH_Left] AND NOT abSharpenStick[PH_Left])  OR NOT abUseSpindle[PH_Left]) AND
								((NOT abChangeStick[PH_Right] AND NOT abSharpenStick[PH_Right])  OR NOT abUseSpindle[PH_Right]) THEN
									alrCurrentSpeed[PA_Z1] := alrMaxRobotSpeed[PA_Z1];
									alrCurrentSpeed[PA_Z2] := alrMaxRobotSpeed[PA_Z2];
									alrTargetPos[PA_Z1] := alrSafePos[PA_Z1];
									alrTargetPos[PA_Z2] := alrSafePos[PA_Z2];
									aeMoveRobotCommand[PA_Z1] := AC_MoveAtAbsPos;
									aeMoveRobotCommand[PA_Z2] := AC_MoveAtAbsPos;
									sCurrentState.eStep := SP_RunStp32;
							END_IF
						SP_RunStp32:
							(* Stop motors *)
							abStartPearlingMotor[PH_Left] := FALSE;
							abStartPearlingMotor[PH_Right] := FALSE;
							(* Move to ref pearl *)
							IF (aTRobotAxis[PA_Z1].eCurrentState = AS_InPosition) AND
									(aTRobotAxis[PA_Z2].eCurrentState = AS_InPosition) THEN
								alrTargetPos[PA_X] := alrPearlingOffset[PA_X]  + sRunData.sPearlingData.aDataPerlage[PH_Left].lrX *alrPearlingInvert[PA_X] ;
								alrTargetPos[PA_Y] := alrPearlingOffset[PA_Y]  + sRunData.sPearlingData.aDataPerlage[PH_Left].lrY *alrPearlingInvert[PA_Y] ;
								aeMoveRobotCommand[PA_X] := AC_MoveAtAbsPos;
								aeMoveRobotCommand[PA_Y] := AC_MoveAtAbsPos;
								sCurrentState.eStep := SP_RunStp33;
							END_IF
						SP_RunStp33:
							IF (eRobotXYStatus = AS_InPosition) THEN
								sCurrentState.bWaitStep := TRUE;
								(* Move to pre ref for probing *)
								FOR iSide := 0 TO 1 DO
									IF abTakeZRef[iSide] THEN
										alrProbingLimit[iSide] :=  alrPearlingOffset[PA_Z1+iSide] + 1.5;
										abDoProbing[iSide] := TRUE;
										abRetryProbing[iSide] := TRUE; (* Part can slide on the layering and stick should not slide in the chuck here, so we can restart a failed probing *)
										aeProbingArea[iSide] := aePearlingArea[iSide];
										alrTargetPos[PA_Z1+iSide] := alrPearlingOffset[PA_Z1+iSide]  - sPartData.lrPartAndLayeringHeight - asStickData[iSide].lrOutLength - 0.5;	// TODO: HFO, change the value, original -1
										aeMoveRobotCommand[PA_Z1+iSide] := AC_MoveAtAbsPos;
									END_IF
								END_FOR
								sCurrentState.eStep := SP_RunStp34;
							END_IF
						SP_RunStp34:
							IF (abProbingDone[PH_Left] OR NOT abTakeZRef[PH_Left]) AND (abProbingDone[PH_Right] OR NOT abTakeZRef[PH_Right]) THEN
								FOR iSide:=0 TO 1 DO
									IF abTakeZRef[iSide] THEN
										alrSecurityPosition[aiPearlingLayringPos[iSide], aiPearlingLayringOffsetPos[iSide], iSide] := alrProbingPos[iSide] - sRunData.sPearlingData.aDataPerlage[PH_Left].lrZ * alrPearlingInvert[PA_Z1+iSide] + sRunData.sPearlingData.lrSecurityZ * alrPearlingInvert[PA_Z1+iSide]  + asStickData[iSide].lrOutLength;
										alrContactPosition[aiPearlingLayringPos[iSide], aiPearlingLayringOffsetPos[iSide], iSide] := alrProbingPos[iSide] - sRunData.sPearlingData.aDataPerlage[PH_Left].lrZ * alrPearlingInvert[PA_Z1+iSide];
										alrContactStickPosition[aiPearlingLayringPos[iSide], aiPearlingLayringOffsetPos[iSide], iSide] := alrContactPosition[aiPearlingLayringPos[iSide], aiPearlingLayringOffsetPos[iSide], iSide] - alrStickCorrection[iSide];
										alrProbingRef[aiPearlingLayringPos[iSide], aiPearlingLayringOffsetPos[iSide], iSide] := alrSharpenProbing[iSide];
										abZRefTaken[aiPearlingLayringPos[iSide], aiPearlingLayringOffsetPos[iSide], iSide] := TRUE;
										alrHeadContactPosition[iSide] := alrContactPosition[aiPearlingLayringPos[iSide], aiPearlingLayringOffsetPos[iSide], iSide];
										alrPreRefPosZ[iSide] := alrHeadContactPosition[iSide] - lrSecurityPreRefPosZ;
										alrTargetPos[PA_Z1+iSide] := alrPreRefPosZ[iSide];
										abTakeZRef[iSide] := FALSE;
										aeMoveRobotCommand[PA_Z1+iSide] := AC_MoveAtAbsPos;
									END_IF
								END_FOR
								sCurrentState.eStep := SP_RunStp35;
							END_IF
						SP_RunStp35:
							IF (aTRobotAxis[PA_Z1].eCurrentState = AS_InPosition) AND
									(aTRobotAxis[PA_Z2].eCurrentState = AS_InPosition) THEN
								FOR iSide:=0 TO 1 DO
									abDoProbing[iSide] := FALSE;
								END_FOR
								(* First move Z to safe *)
(*								alrTargetPos[PA_Z1] := alrSafePos[PA_Z1];
								alrTargetPos[PA_Z2] := alrSafePos[PA_Z2];
								aeMoveRobotCommand[PA_Z1] := AC_MoveAtAbsPos;
								aeMoveRobotCommand[PA_Z2] := AC_MoveAtAbsPos;
*)								sCurrentState.bWaitStep := TRUE;
								sCurrentState.eStep := SP_RunStp7;
							END_IF
						SP_RunStp40:
							(* We are ready for pearling, mark part for reject is something goes wrong *)
							FOR iSide := 0 TO 1 DO
								IF abUseSpindle[iSide] THEN
									sRunData.apsPartData[iSide]^.abHasPearls[aiSideInfo[iSide],sRunData.apsPartData[iSide]^.ePartSide] := TRUE;
								END_IF
							END_FOR
							sCurrentState.eStep := SP_RunStp41;
						SP_RunStp41:
							(* Get pearling parameter *)
							FOR iSide:=0 TO 1 DO
								alrHeadSecurityPosition[iSide] := alrSecurityPosition[aiPearlingLayringPos[iSide], aiPearlingLayringOffsetPos[iSide], iSide];
								alrHeadContactPosition[iSide] := alrContactPosition[aiPearlingLayringPos[iSide], aiPearlingLayringOffsetPos[iSide], iSide];
								alrPreRefPosZ[iSide] := alrHeadContactPosition[iSide] - lrSecurityPreRefPosZ;
								alrHeadProbingRef[iSide] := alrProbingRef[aiPearlingLayringPos[iSide], aiPearlingLayringOffsetPos[iSide], iSide];
								alrHeadContactStickPosition[iSide] := alrContactStickPosition[aiPearlingLayringPos[iSide], aiPearlingLayringOffsetPos[iSide], iSide];
							END_FOR
							sCurrentState.eStep := SP_RunStp50;
						SP_RunStp50:
							IF (aTRobotAxis[PA_Z1].eCurrentState = AS_InPosition) AND
									(aTRobotAxis[PA_Z2].eCurrentState = AS_InPosition) THEN
								bEndPearling := TRUE;
								FOR iSide:=0 TO 1 DO
									IF abUseSpindle[iSide] THEN
										IF NOT sRunData.apsPartData[iSide]^.abPearlingDone[aiSideInfo[iSide],sRunData.apsPartData[iSide]^.ePartSide] THEN
											bEndPearling := FALSE;
										END_IF
									END_IF
								END_FOR
								IF bEndPearling THEN
									(* End of pearling *)
									sCurrentState.eStep := SP_RunStp80;
								END_IF
								WHILE( sCurrentState.eStep = SP_RunStp50) DO
									IF (nPearlIndex < sRunData.sPearlingData.nNbOfPearls) THEN
										(* Continue with next pearl *)
										IF sRunData.sPearlingData.aDataPerlage[nPearlIndex].bDisable THEN
											nPearlIndex := nPearlIndex + 1;
										ELSE
											sCurrentState.bWaitStep := TRUE;
											sCurrentState.eStep := SP_RunStp51;
										END_IF
									ELSE
										(* End of pearling *)
										sCurrentState.eStep := SP_RunStp80;
									END_IF
								END_WHILE
							END_IF
						SP_RunStp51:
							(* Check if a sharpen is needed *)
							FOR iSide:=0 TO 1 DO
								abNeedSharpening[iSide] := FALSE;
							END_FOR
							IF (iCurrentArea <> sRunData.sPearlingData.aDataPerlage[nPearlIndex].iArea) THEN
								(* We change area, check if we can do the entire area without sharpening *)
								iCurrentArea := sRunData.sPearlingData.aDataPerlage[nPearlIndex].iArea;
								FOR iSide:=0 TO 1 DO
									IF  sRunData.sPearlingData.iSharpenFreq > 0 AND aArea[iCurrentArea].iNbOfPearls + aiNbOfPearlsDone[iSide] > sRunData.sPearlingData.iSharpenFreq AND abUseSpindle[iSide] THEN
										abNeedSharpening[iSide] := TRUE;
									END_IF
								END_FOR
							END_IF
							FOR iSide:=0 TO 1 DO
								(* Check if sharpen need if Area is bigger then SharpenFreq, should not happen *)
								IF  sRunData.sPearlingData.iSharpenFreq > 0 AND aiNbOfPearlsDone[iSide] > sRunData.sPearlingData.iSharpenFreq  AND abUseSpindle[iSide] THEN
									abNeedSharpening[iSide] := TRUE;
								END_IF
								(* Check force sharpen for each pearl *)
								IF sRunData.sPearlingData.aDataPerlage[nPearlIndex].bForceSharpen  AND abUseSpindle[iSide] THEN
									abNeedSharpening[iSide] := TRUE;
								END_IF
							END_FOR
							IF ((abNeedSharpening[PH_Left] OR abNeedChangeStick[PH_Left]) AND abUseSpindle[PH_Left]) OR
								((abNeedSharpening[PH_Right] OR abNeedChangeStick[PH_Right]) AND abUseSpindle[PH_Right]) THEN
								sCurrentState.eStep := SP_RunStp52;
							ELSE
								sCurrentState.eStep := SP_RunStp54;
							END_IF
						SP_RunStp52 :
							(* Sharpen stick *)
							FOR iSide:=0 TO 1 DO
								IF abUseSpindle[iSide] THEN
									IF abNeedSharpening[iSide] AND NOT abNeedChangeStick[iSide] THEN
										abSharpenStick[iSide] := TRUE;
									END_IF
									IF abNeedChangeStick[iSide] THEN
										abChangeStick[iSide] := TRUE;
										abNeedChangeStick[iSide] := FALSE;
									END_IF
								END_IF
							END_FOR
							sCurrentState.eStep := SP_RunStp53;
						SP_RunStp53 :
							(* Wait end of sharpening during prod *)
							IF ((NOT abChangeStick[PH_Left] AND NOT abSharpenStick[PH_Left])  OR NOT abUseSpindle[PH_Left]) AND
								((NOT abChangeStick[PH_Right] AND NOT abSharpenStick[PH_Right])  OR NOT abUseSpindle[PH_Right]) THEN
								(* Move Z to safe *)
								FOR iSide:=0 TO 1 DO
									alrTargetPos[PA_Z1+iSide] := alrSafePos[PA_Z1+iSide];
									aeMoveRobotCommand[PA_Z1+iSide] := AC_MoveAtAbsPos;
								END_FOR
								sCurrentState.eStep := SP_RunStp54;
							END_IF
						SP_RunStp54:
							(* Do one pearl *)
							IF bPauseReq THEN
								(* Stop request during prod*)
								FOR iSide:=0 TO 1 DO
									abPearlingWeightOutOfToleranceDetected[iSide] := FALSE;
									abStickBrokenDetected[iSide] := FALSE;
								END_FOR
								bSecurityErrorDetected := FALSE;
								sCurrentState.eStep := SP_RunStp90;
							ELSE
								(* Security already checked before pearling start*)
								(* Move to preref pos if needed *)
								IF sRunData.sPearlingData.aDataPerlage[nPearlIndex].bMoveToSafe THEN
									FOR iSide:=0 TO 1 DO
										IF abUseSpindle[iSide] THEN
											alrTargetPos[PA_Z1+iSide] := alrPreRefPosZ[iSide];
											aeMoveRobotCommand[PA_Z1+iSide] := AC_MoveAtAbsPos;
										END_IF
									END_FOR
								END_IF
								sCurrentState.eStep := SP_RunStp55;
							END_IF
						SP_RunStp55:
							IF (aTRobotAxis[PA_Z1].eCurrentState = AS_InPosition) AND (aTRobotAxis[PA_Z2].eCurrentState = AS_InPosition) THEN
								(* Move to XY pearl *)
								FOR iSide:=0 TO 1 DO
									aTDispersion[iSide](bGenerate := TRUE, nPearl := nPearlIndex );
								END_FOR
								alrTargetPos[PA_X] := alrPearlingOffset[PA_X]  + sRunData.sPearlingData.aDataPerlage[nPearlIndex].lrX *alrPearlingInvert[PA_X];
								alrTargetPos[PA_Y] := alrPearlingOffset[PA_Y]  + sRunData.sPearlingData.aDataPerlage[nPearlIndex].lrY *alrPearlingInvert[PA_Y];
								IF (sRunData.sPearlingData.aDataPerlage[nPearlIndex].bXYDispersion) THEN
									alrTargetPos[PA_X] := alrTargetPos[PA_X]  + ((aTDispersion[PH_Left].lrDispersionX * INT_TO_LREAL(sRunData.sPearlingData.iDispersionXY) / 100.0)) - 0.5;
									alrTargetPos[PA_Y] := alrTargetPos[PA_Y]  + ((aTDispersion[PH_Left].lrDispersionY * INT_TO_LREAL(sRunData.sPearlingData.iDispersionXY) / 100.0)) - 0.5;
								END_IF
								aeMoveRobotCommand[PA_X] := AC_MoveAtAbsPos;
								aeMoveRobotCommand[PA_Y] := AC_MoveAtAbsPos;
								sCurrentState.eStep := SP_RunStp60;
							END_IF
						SP_RunStp60 :
							IF (eRobotXYStatus = AS_InPosition) THEN
								FOR iSide:=0 TO 1 DO
									IF abUseSpindle[iSide] THEN
										aeProbingArea[iSide] := aePearlingArea[iSide]; (* redefine probing area, could be change by sharpening *)
										alrTargetPos[PA_Z1+iSide] := alrPreRefPosZ[iSide];
										aeMoveRobotCommand[PA_Z1+iSide] := AC_MoveAtAbsPos;
									END_IF
								END_FOR
								sCurrentState.eStep := SP_RunStp61;
							END_IF
						SP_RunStp61 :
							IF (eRobotXYStatus = AS_InPosition) AND (aTRobotAxis[PA_Z1].eCurrentState = AS_InPosition) AND (aTRobotAxis[PA_Z2].eCurrentState = AS_InPosition) AND
								NOT asPearlData[PH_Left].bNewPearl AND NOT asPearlData[PH_Right].bNewPearl AND NOT asPearlData[PH_Left].bNewPart AND NOT asPearlData[PH_Right].bNewPart
								AND (aTWaitMotorStarted[PH_Left].Q OR  NOT abUseSpindle[PH_Left]) AND (aTWaitMotorStarted[PH_Right].Q OR  NOT abUseSpindle[PH_Right]) THEN
								(* Calculate pearl energy with dispersion *)
								IF (sRunData.sPearlingData.aDataPerlage[nPearlIndex].lrRate > 100) THEN
									sRunData.sPearlingData.aDataPerlage[nPearlIndex].lrRate := 100;
								END_IF
								bSecurityErrorDetected := FALSE;
								FOR iSide:=0 TO 1 DO
									abStickBrokenDetected[iSide] := FALSE;
									abPearlingWeightOutOfToleranceDetected[iSide] := FALSE;
									IF abUseSpindle[iSide] THEN
										abPearlNeeded[iSide] := nPearlIndex > anPearlIndexDone[iSide] AND NOT sRunData.apsPartData[iSide]^.abPearlingDone[aiSideInfo[iSide],sRunData.apsPartData[iSide]^.ePartSide];
										IF nPearlIndex < anPearlIndexDone[iSide] THEN
											nPearlIndex := anPearlIndexDone[iSide] + 1;
										END_IF
									ELSE
										abPearlNeeded[iSide] := FALSE;
									END_IF
									IF abPearlNeeded[iSide] THEN
										alrDeltaSharpenProbing[iSide] := (alrSharpenProbing[iSide] - alrHeadProbingRef[iSide]) * 1000;
										alrPearlingEnergy[iSide] := alrBasePearlingEnergy[iSide] * (1-((aTDispersion[iSide].lrDispersionZ * INT_TO_LREAL(sRunData.sPearlingData.iDispersionZ))/100))*(sRunData.sPearlingData.aDataPerlage[nPearlIndex].lrRate/100)*alrRatiog2mm[iSide];
										(* Do pearl, first move Z to position with correction *)
										abCheckingStick[iSide] := (alrPearlingEnergy[iSide] >= 0.07);
										alrTargetPos[PA_Z1+iSide] := alrHeadContactPosition[iSide] + sRunData.sPearlingData.aDataPerlage[nPearlIndex].lrZ* alrPearlingInvert[PA_Z1+iSide] + alrPearlingEnergy[iSide] + alrCorrectionMCR[iSide];
										alrDeltaStickCorrection[iSide] := alrTargetPos[PA_Z1+iSide] - (alrHeadContactStickPosition[iSide] + sRunData.sPearlingData.aDataPerlage[nPearlIndex].lrZ* alrPearlingInvert[PA_Z1+iSide] + alrPearlingEnergy[iSide] + alrCorrectionMCR[iSide] + alrStickCorrection[iSide]);
										(*alrTargetPos[PA_Z1+iSide] := alrHeadContactStickPosition[iSide] + sRunData.sPearlingData.aDataPerlage[nPearlIndex].lrZ* alrPearlingInvert[PA_Z1+iSide] + alrPearlingEnergy[iSide] + alrCorrectionMCR[iSide] + alrStickCorrection[iSide]; *)
										alrTargetPos[PA_Z1+iSide] := alrTargetPos[PA_Z1+iSide] + alrDeltaStickCorrection[iSide];
										(*alrDeltaStickCorrection[iSide] := alrHeadContactPosition[iSide] - alrHeadContactStickPosition[iSide] - alrStickCorrection[iSide];*)
										IF (alrTargetPos[PA_Z1+iSide] > alrHeadSecurityPosition[iSide]) THEN
											(* this part is aborted and mark for reject *)
											sRunData.apsPartData[iSide]^.abBadPearling[iSide,sRunData.apsPartData[iSide]^.ePartSide] := TRUE;
											sRunData.apsPartData[iSide]^.abPearlingDone[aiSideInfo[iSide],sRunData.apsPartData[iSide]^.ePartSide] := TRUE;
											bSecurityErrorDetected := TRUE;
											iDebugPos := 5;
											iDebugSide := iSide;
										ELSE
											aeMoveRobotCommand[PA_Z1+iSide] := AC_MoveAtAbsPos;
											abPearlStarted[iSide] := FALSE;
											abPearlDone[iSide] := FALSE;
											abPearlPosReached[iSide] := FALSE;
											aIMinPos[iSide] := 32767;
											sCurrentState.eStep := SP_RunStp62;
										END_IF
									END_IF
								END_FOR
								FOR iSide:=0 TO 1 DO
									IF abPearlNeeded[iSide] AND NOT bSecurityErrorDetected THEN
										abBadPearling[iSide] := sRunData.apsPartData[iSide]^.abBadPearling[iSide,sRunData.apsPartData[iSide]^.ePartSide];
										sRunData.apsPartData[iSide]^.abBadPearling[iSide,sRunData.apsPartData[iSide]^.ePartSide] := TRUE;
									END_IF
								END_FOR
							END_IF
							IF bSecurityErrorDetected THEN
								aeMoveRobotCommand[PA_Z1] := AC_None;
								aeMoveRobotCommand[PA_Z2] := AC_None;
								sCurrentState.eStep := SP_RunStp90;
							END_IF
						SP_RunStp62: (* Do pearl here *)
							FOR iSide:=0 TO 1 DO
								IF abPearlNeeded[iSide] THEN
									IF NOT abPearlStarted[iSide] AND ((aTRobotAxis[PA_Z1+iSide].lrCurrentPos > (alrHeadContactPosition[iSide] + sRunData.sPearlingData.aDataPerlage[nPearlIndex].lrZ * alrPearlingInvert[PA_Z1+iSide]))  OR aTRobotAxis[PA_Z1+iSide].eCurrentState = AS_InPosition) THEN
										aTDetectStickBroken[iSide](IN := FALSE);
										aTPearlingTimer[iSide](IN := FALSE);
										abPearlStarted[iSide] := TRUE;
									END_IF
									IF abPearlStarted[iSide] AND NOT abPearlDone[iSide] THEN
										aTPearlingTimer[iSide](IN := TRUE,PT := INT_TO_TIME(sRunData.sPearlingData.iPearlingTime));
										aTDetectStickBroken[iSide](IN := NOT abStickContact[iSide] AND abCheckingStick[iSide] AND (aTRobotAxis[PA_Z1+iSide].eCurrentState = AS_InPosition),PT := TBreakStickDetectTime);
										IF aTDetectStickBroken[iSide].Q AND NOT abPearlDone[iSide] THEN
											abStickBrokenDetected[iSide] := TRUE;
											iDebugPosBrokenStick := 10;
											iDebugSide := iSide;
										END_IF
										IF aTRobotAxis[PA_Z1+iSide].eCurrentState = AS_InPosition OR aTPearlingTimer[iSide].Q THEN
											abPearlPosReached[iSide] := TRUE;
											IF aiContactDistance[iSide] < aIMinPos[iSide] THEN
												aIMinPos[iSide] := aiContactDistance[iSide];
											END_IF
										END_IF
										IF aTPearlingTimer[iSide].Q THEN
											(* Move Z to pre-ref *)
											abPearlDone[iSide] := TRUE;
											aiNbOfPearlsDone[iSide] := aiNbOfPearlsDone[iSide] + 1;
											(* pearling speed optimization in counterbores *)
											IF bUsePearlMoveToSafe THEN
												alrTargetPos[PA_Z1+iSide] := alrHeadContactPosition[iSide] + sRunData.sPearlingData.aDataPerlage[nPearlIndex].lrZ* alrPearlingInvert[PA_Z1+iSide] - lrSecurityPreRefPosZ;
											ELSE
												alrTargetPos[PA_Z1+iSide] := alrPreRefPosZ[iSide];
											END_IF
											aeMoveRobotCommand[PA_Z1+iSide] := AC_MoveAtAbsPos;
										END_IF
									END_IF
								ELSE
									abPearlDone[iSide] := TRUE;
								END_IF
							END_FOR
							IF (abPearlDone[PH_Left]  AND abPearlDone[PH_Right]) THEN
								FOR iSide:=0 TO 1 DO
									IF abPearlNeeded[iSide] THEN
										alrDeltaZPearl[iSide] :=INT_TO_LREAL(aIMinPos[iSide] - aiContactThresholdArea[iSide , aePearlingArea[iSide]]) / alrSensorRate[iSide];
										alrDeltaWeightPearl[iSide] := (alrPearlingEnergy[iSide] - alrDeltaZPearl[iSide]) / alrRatiog2mm[iSide];
										asPearlData[iSide].iPearlNb := UINT_TO_INT(nPearlIndex);
										asPearlData[iSide].iRate := DINT_TO_INT(TRUNC((sRunData.sPearlingData.aDataPerlage[nPearlIndex].lrRate+0.1)));
										asPearlData[iSide].lrDispersion := aTDispersion[iSide].lrDispersionZ * INT_TO_LREAL(sRunData.sPearlingData.iDispersionZ);
										asPearlData[iSide].lrPearlingCalcPos := alrPearlingEnergy[iSide];
										asPearlData[iSide].lrCorrectionMCR := alrCorrectionMCR[iSide];
										asPearlData[iSide].lrDeltaCurrent := 0;(*TMCRDrv.lrPower; *)
										asPearlData[iSide].lrPearlingMeasurePos := 0;(* TMCRDrv.lrPower*sStickData.sStickDataMMI.lrMA2MMFactor;*)
										asPearlData[iSide].lrSensorProbePos := alrHeadContactPosition[iSide];
										asPearlData[iSide].lrSensorPearlPos := alrDeltaZPearl[iSide];
										asPearlData[iSide].lrDeltaWeight := alrDeltaWeightPearl[iSide];
										asPearlData[iSide].bNewPearl := TRUE;
										asPearlData[iSide].iVacuumFlow := aiVacuumFlow[iSide];
										adwPearlsCounter[iSide] := adwPearlsCounter[iSide] + 1;
									END_IF
								END_FOR
								sCurrentState.eStep := SP_RunStp63;
							END_IF
						SP_RunStp63:
							IF (aTRobotAxis[PA_Z1].eCurrentState = AS_InPosition) AND (aTRobotAxis[PA_Z2].eCurrentState = AS_InPosition) THEN
								FOR iSide:=0 TO 1 DO
									IF abPearlNeeded[iSide] THEN
										 (* Check if pearl has been process correctly *)
										IF ((alrPearlingEnergy[iSide] - alrDeltaZPearl[iSide] + alrCorrectionMCR[iSide]) > lrStickErrorDeltaPos) THEN
											abStickBrokenDetected[iSide] := TRUE;
											iDebugPosBrokenStick := 11;
											iDebugSide := iSide;
										END_IF
										IF ABS(alrDeltaWeightPearl[iSide]) >= sStickDataShared.sStickDataMMIShared.iWeightTolerance THEN
											abPearlingWeightOutOfToleranceDetected[iSide] := TRUE;
										END_IF
										IF NOT abStickBrokenDetected[iSide] AND NOT abPearlingWeightOutOfToleranceDetected[iSide] THEN
											anPearlIndexDone[iSide] := nPearlIndex;
											sRunData.apsPartData[iSide]^.anLastPearlIndexDone[aiSideInfo[iSide],sRunData.apsPartData[iSide]^.ePartSide] := nPearlIndex;
										END_IF
										IF abStickBrokenDetected[iSide] OR abPearlingWeightOutOfToleranceDetected[iSide] THEN
											abBadPearling[iSide] := TRUE;
										END_IF
										sRunData.apsPartData[iSide]^.abBadPearling[iSide,sRunData.apsPartData[iSide]^.ePartSide] := abBadPearling[iSide];
										 (* Calculate correction *)
										lrMaxMCRCorrection := asStickDataMMI[iSide].lrMCRCorrectionStep;
										IF abFirstPearl[iSide] THEN
											lrMaxMCRCorrection := 0.2;
											alrFirstPearlCorrection[iSide] := (alrDeltaZPearl[iSide] - alrPearlingEnergy[iSide]) * 1000;
											abFirstPearl[iSide] := FALSE;
										END_IF
										IF  (alrDeltaZPearl[iSide] > alrPearlingEnergy[iSide]) THEN
											IF ABS(alrDeltaZPearl[iSide] - alrPearlingEnergy[iSide]) > lrMaxMCRCorrection THEN
												alrCorrectionMCR[iSide] := alrCorrectionMCR[iSide] - lrMaxMCRCorrection;
											ELSE
												alrCorrectionMCR[iSide] := alrCorrectionMCR[iSide] - ABS(alrDeltaZPearl[iSide] - alrPearlingEnergy[iSide]);
											END_IF
										ELSIF (alrDeltaZPearl[iSide] < alrPearlingEnergy[iSide]) THEN
											IF ABS(alrDeltaZPearl[iSide] - alrPearlingEnergy[iSide]) > lrMaxMCRCorrection THEN
												alrCorrectionMCR[iSide] := alrCorrectionMCR[iSide] + lrMaxMCRCorrection;
											ELSE
												alrCorrectionMCR[iSide] := alrCorrectionMCR[iSide] + ABS(alrDeltaZPearl[iSide] - alrPearlingEnergy[iSide]);
											END_IF
										END_IF
									END_IF
								END_FOR
								sCurrentState.eStep := SP_RunStp64;
							END_IF
						SP_RunStp64: (* Error management *)
							IF abStickBrokenDetected[PH_Left] OR abStickBrokenDetected[PH_Right] OR abPearlingWeightOutOfToleranceDetected[PH_Left] OR abPearlingWeightOutOfToleranceDetected[PH_Right] THEN
								FOR iSide:=0 TO 1 DO
									IF abPearlNeeded[iSide] THEN
										IF sStickDataShared.sStickDataMMIShared.bRestartBeginOfArea AND abStickBrokenDetected[iSide] THEN
											nPearlIndex := INT_TO_UINT(aArea[iCurrentArea].iFirstPearl);
											anPearlIndexDone[iSide] := nPearlIndex;
											sRunData.apsPartData[iSide]^.anLastPearlIndexDone[aiSideInfo[iSide],sRunData.apsPartData[iSide]^.ePartSide] := nPearlIndex;
										END_IF
										IF abStickBrokenDetected[iSide] OR abPearlingWeightOutOfToleranceDetected[iSide] THEN
											aiCountPearlError[iSide] := aiCountPearlError[iSide] + 1;
										END_IF
										IF abStickBrokenDetected[iSide] OR abPearlingWeightOutOfToleranceDetected[iSide] THEN
											aiCountPearlError[iSide] := aiCountPearlError[iSide] + 1;
										END_IF
										IF sStickDataShared.sStickDataMMIShared.bStopOnStickBreak AND abStickBrokenDetected[iSide] THEN
											aiCountPearlError[iSide] := 3;
										END_IF
										IF sStickDataShared.sStickDataMMIShared.bStopOnWeightOutOfTolerance AND abPearlingWeightOutOfToleranceDetected[iSide] THEN
											aiCountPearlError[iSide] := 3;
										END_IF
									END_IF
								END_FOR
								IF (aiCountPearlError[PH_Left] >= 3 AND abPearlNeeded[PH_Left]) OR (aiCountPearlError[PH_Right] >= 3 AND abPearlNeeded[PH_Right]) THEN
									FOR iSide:=0 TO 1 DO
										IF abPearlNeeded[iSide] AND aiCountPearlError[iSide] >= 3 THEN
											aiCountPearlError[iSide] := 0;
										END_IF
									END_FOR
									sCurrentState.eStep := SP_RunStp90; (* Stop during process *)
								ELSE
									sCurrentState.eStep := SP_RunStp50; (* continue process *)
								END_IF
							ELSE
								(* Check next pearl *)
								nPearlIndex := nPearlIndex + 1;
								sCurrentState.eStep := SP_RunStp50;
							END_IF
						SP_RunStp80:
							(* Pearling is finished *)
							(* Move Z to safe *)
							alrTargetPos[PA_Z1] := alrSafePos[PA_Z1];
							alrTargetPos[PA_Z2] := alrSafePos[PA_Z2];
							aeMoveRobotCommand[PA_Z1] := AC_MoveAtAbsPos;
							aeMoveRobotCommand[PA_Z2] := AC_MoveAtAbsPos;
							sCurrentState.eStep := SP_RunStp81;
						SP_RunStp81:
							IF (aTRobotAxis[PA_Z1].eCurrentState = AS_InPosition) AND
									(aTRobotAxis[PA_Z2].eCurrentState = AS_InPosition) THEN
								FOR iSide:=0 TO 1 DO
									abAspirationPearling[iSide] := FALSE;
									IF abUseSpindle[iSide] THEN
										sRunData.apsPartData[iSide]^.abPearlingDone[aiSideInfo[iSide],sRunData.apsPartData[iSide]^.ePartSide] := TRUE;
										aTDispersion[iSide](bNewPart := TRUE);
										//sRunData.apsPartData[iSide]^.bToReject := sRunData.apsPartData[iSide]^.bToReject OR sRunData.apsPartData[iSide]^.abBadPearling[0,0] OR sRunData.apsPartData[iSide]^.abBadPearling[0,1] OR sRunData.apsPartData[iSide]^.abBadPearling[PH_Right,0] OR sRunData.apsPartData[iSide]^.abBadPearling[1,1];
										sRunData.apsPartData[iSide]^.bToReject := sRunData.apsPartData[iSide]^.abBadPearling[PH_Left,PS_SUS] OR sRunData.apsPartData[iSide]^.abBadPearling[PH_Left,PS_SOUS] OR sRunData.apsPartData[iSide]^.abBadPearling[PH_Right,PS_SUS] OR sRunData.apsPartData[iSide]^.abBadPearling[PH_Right,PS_SOUS];
									END_IF
								END_FOR
								(* Force a sharpen if needed *)
								IF sRunData.bForceSharpenAfterPearling THEN
									abUseSpindle := abHeadIsUsed;
									FOR iSide:=0 TO 1 DO
										abSharpenStick[iSide] := TRUE;
									END_FOR
								ELSE (*IF abUseSpindle[0] AND abUseSpindle[1] THEN*)
									iCurrentArea := sRunData.sPearlingData.aDataPerlage[PH_Right].iArea;
									FOR iSide:=0 TO 1 DO
										IF  abUseSpindle[iSide] THEN
											IF sRunData.sPearlingData.iSharpenFreq > 0 AND ((aiNbOfPearlsDone[iSide] + aArea[iCurrentArea].iNbOfPearls) > sRunData.sPearlingData.iSharpenFreq) THEN
												abSharpenStick[iSide] := TRUE;
											END_IF
											IF sRunData.sPearlingData.aDataPerlage[PH_Right].bForceSharpen THEN
												abSharpenStick[iSide] := TRUE;
											END_IF
										END_IF
									END_FOR
									IF bParallelProduction AND (abSharpenStick[PH_Left] OR abSharpenStick[PH_Right]) THEN
										(* Sharpen both head if we are in parrelle mode *)
										abUseSpindle := abHeadIsUsed;
										abSharpenStick[PH_Left] := TRUE;
										abSharpenStick[PH_Right] := TRUE;
									END_IF
								END_IF
								sCurrentState.eStep := SP_RunStp1;
							END_IF
						SP_RunStp90:
							(* Stop request during pearling, move to safe *)
							FOR iSide := 0 TO 1 DO
								alrTargetPos[PA_Z1+iSide] := alrSafePos[PA_Z1+iSide];
								aeMoveRobotCommand[PA_Z1+iSide] := AC_MoveAtAbsPos;
							END_FOR
							sCurrentState.eStep := SP_RunStp91;
						SP_RunStp91:
							IF (aTRobotAxis[PA_Z1].eCurrentState = AS_InPosition) AND
									(aTRobotAxis[PA_Z2].eCurrentState = AS_InPosition) THEN
								FOR iSide := 0 TO 1 DO
									IF abPearlingWeightOutOfToleranceDetected[iSide] THEN
										abPearlingWeightOutOfToleranceError[iSide] := TRUE;
										abSharpenStick[iSide] := TRUE;
										abTakeZRef[iSide] := TRUE;
									END_IF
									abPearlingWeightOutOfToleranceDetected[iSide] := FALSE;
									IF abStickBrokenDetected[iSide] THEN
										abStickBroken[iSide] := TRUE;
										abNeedChangeStick[iSide] := TRUE;
									END_IF
									abStickBrokenDetected[iSide] := FALSE;
									IF abNeedChangeStick[iSide] THEN
										abChangeStick[iSide] := TRUE;
										abTakeZRef[iSide] := TRUE;
									END_IF
									abNeedChangeStick[iSide] := FALSE;
								END_FOR
								IF bSecurityErrorDetected THEN
									bSecurityError := TRUE;
								END_IF
								bSecurityErrorDetected := FALSE;
								(* Stop module *)
								sCurrentState.eStep := SP_RunStp92;
							END_IF
						SP_RunStp92:
							IF ((NOT abChangeStick[PH_Left] AND NOT abSharpenStick[PH_Left])  OR NOT abUseSpindle[PH_Left]) AND
									((NOT abChangeStick[PH_Right] AND NOT abSharpenStick[PH_Right])  OR NOT abUseSpindle[PH_Right]) THEN
								sCurrentState.eStep := SP_RunStp30;
							END_IF
						SP_RunStp200:(* Change Chuck *)
							IF ((NOT abChangeStick[PH_Left] AND NOT abSharpenStick[PH_Left])  OR NOT abUseSpindle[PH_Left]) AND
								((NOT abChangeStick[PH_Right] AND NOT abSharpenStick[PH_Right])  OR NOT abUseSpindle[PH_Right]) THEN
								FOR iSide:=0 TO 1 DO
									abUseSpindle[iSide] := FALSE;
								END_FOR
								alrCurrentSpeed := alrMaxRobotSpeed;
								alrTargetPos[PA_Z1] := alrSafePos[PA_Z1];
								alrTargetPos[PA_Z2] := alrSafePos[PA_Z2];
								aeMoveRobotCommand[PA_Z1] := AC_MoveAtAbsPos;
								aeMoveRobotCommand[PA_Z2] := AC_MoveAtAbsPos;
								sCurrentState.eStep := SP_RunStp201;
							END_IF
						SP_RunStp201 :
							IF 	(aTRobotAxis[PA_Z1].eCurrentState = AS_InPosition) AND
								(aTRobotAxis[PA_Z2].eCurrentState = AS_InPosition) THEN
								IF bChangeToolSide THEN
									alrTargetPos[PA_X] := aTRobotAxis[PA_X].lrMinPos+1;
									alrTargetPos[PA_Y] := aTRobotAxis[PA_Y].lrMinPos+1;
								ELSE
									alrTargetPos[PA_X] := aTRobotAxis[PA_X].lrMaxPos-1;
									alrTargetPos[PA_Y] := aTRobotAxis[PA_Y].lrMinPos+1;
								END_IF
								bChangeToolSide := NOT bChangeToolSide;
								aeMoveRobotCommand[PA_X] := AC_MoveAtAbsPos;
								aeMoveRobotCommand[PA_Y] := AC_MoveAtAbsPos;
								sCurrentState.eStep := SP_RunStp202;
							END_IF
						SP_RunStp202 :
							IF (eRobotXYStatus = AS_InPosition) THEN
								sCurrentState.eStep := SP_RunStp1;
							END_IF
						SP_RunStp210:(* Check Sharpen *)
							IF ((NOT abChangeStick[PH_Left] AND NOT abSharpenStick[PH_Left])  OR NOT abUseSpindle[PH_Left]) AND
								((NOT abChangeStick[PH_Right] AND NOT abSharpenStick[PH_Right])  OR NOT abUseSpindle[PH_Right]) THEN
									sCurrentState.eStep := SP_RunStp211;
							END_IF
						SP_RunStp211: (* it's now safe to switch head used *)
							abUseSpindle := abHeadIsUsed;
							FOR iSide:=0 TO 1 DO
								IF NOT abChuckClosed[iSide] AND abUseSpindle[iSide] THEN
									abChangeStick[iSide] := TRUE;
								END_IF
							END_FOR
							sCurrentState.eStep := SP_RunStp1;
					END_CASE
				END_IF
			MS_Manual :
				CASE eTableSideForLoader OF
					TS_A:
						TManualCmd.eTableSide := TS_B;
					TS_B:
						TManualCmd.eTableSide := TS_A;
					ELSE
						TManualCmd.eTableSide := eTableSideForLoader;
				END_CASE
				TManualCmd.bAxisZSafe[PH_Left] := (aTRobotAxis[PA_Z1].lrCurrentPos < (alrSafePos[PA_Z1]+lrSafeTolerance)) AND ((aTRobotAxis[PA_Z1].eCurrentState = AS_InPosition) OR (aTRobotAxis[PA_Z1].eCurrentState = AS_PowerOff)) AND (aTRobotAxis[PA_Z1].bAxisHomed);
				TManualCmd.bAxisZSafe[PH_Right] := (aTRobotAxis[PA_Z2].lrCurrentPos < (alrSafePos[PA_Z2]+lrSafeTolerance)) AND ((aTRobotAxis[PA_Z2].eCurrentState = AS_InPosition) OR (aTRobotAxis[PA_Z2].eCurrentState = AS_PowerOff)) AND (aTRobotAxis[PA_Z2].bAxisHomed);;

				TManualCmd.aTStartMotor[PH_Left].Enable :=  bPowerOn AND NOT abOpenChuck[PH_Left];
				TManualCmd.aTOpenChuck[PH_Left].Enable := NOT abStartPearlingMotor[PH_Left];
				TManualCmd.aTStartMotor[PH_Right].Enable :=  bPowerOn AND NOT abOpenChuck[PH_Right];
				TManualCmd.aTOpenChuck[PH_Right].Enable := NOT abStartPearlingMotor[PH_Right];

				bManualZIsSafe :=  (aTRobotAxis[LA_Z1].lrCurrentPos < (alrSafePos[PA_Z1]+lrSafeTolerance)) AND (aTRobotAxis[PA_Z2].lrCurrentPos < (alrSafePos[LA_Z2]+lrSafeTolerance))
						AND (aTRobotAxis[PA_Z1].bAxisHomed) AND (aTRobotAxis[PA_Z2].bAxisHomed);

				TManualCmd.TSafe.Enable := TRUE;
				TManualCmd.aTCalibrateWeight[PH_Left].Enable := NOT bCalibrationInProgress ;
				TManualCmd.aTCalibrateWeight[PH_Right].Enable := NOT bCalibrationInProgress;
				FOR iAxis := 0 TO 3 DO
					TManualCmd.aTCalibrateWeight[PH_Left].Enable := TManualCmd.aTCalibrateWeight[PH_Left].Enable AND aTRobotAxis[iAxis].eCurrentState = AS_InPosition;
					TManualCmd.aTCalibrateWeight[PH_Right].Enable := TManualCmd.aTCalibrateWeight[PH_Right].Enable AND aTRobotAxis[iAxis].eCurrentState = AS_InPosition;
					TManualCmd.TSafe.Enable := TManualCmd.TSafe.Enable AND ((aTRobotAxis[iAxis].eCurrentState = AS_InPosition) OR  (aTRobotAxis[iAxis].eCurrentState = AS_PowerOff)  OR  (aTRobotAxis[iAxis].eCurrentState = AS_NotHomed));
					TManualCmd.aTAxis[iAxis].Home.Enable := ((aTRobotAxis[iAxis].eCurrentState = AS_InPosition) OR (aTRobotAxis[iAxis].eCurrentState = AS_NotHomed));
					TManualCmd.aTAxis[iAxis].MoveBw.Enable := (aTRobotAxis[iAxis].eCurrentState = AS_InPosition) AND ((aTRobotAxis[iAxis].lrCurrentPos - alrJogStep[iAxis] >= aTRobotAxis[iAxis].lrMinPos) OR NOT aTRobotAxis[iAxis].bMinPosMonitoring);
					TManualCmd.aTAxis[iAxis].MoveFw.Enable := (aTRobotAxis[iAxis].eCurrentState = AS_InPosition) AND ((aTRobotAxis[iAxis].lrCurrentPos + alrJogStep[iAxis] <= aTRobotAxis[iAxis].lrMaxPos) OR NOT aTRobotAxis[iAxis].bMaxPosMonitoring);
					TManualCmd.aTAxisPos[iAxis].MoveToTeach.Enable := (aTRobotAxis[iAxis].eCurrentState = AS_InPosition) AND
							(( alrRobotPos[iAxis, TManualCmd.e_TeachPos] >= aTRobotAxis[iAxis].lrMinPos) OR NOT aTRobotAxis[iAxis].bMinPosMonitoring) AND
							((alrRobotPos[iAxis, TManualCmd.e_TeachPos] <= aTRobotAxis[iAxis].lrMaxPos) OR NOT aTRobotAxis[iAxis].bMaxPosMonitoring);
					TManualCmd.aTAxis[iAxis].CurrentPos := aTRobotAxis[iAxis].lrCurrentPos;
					TManualCmd.aTAxisPos[iAxis].TeachedPos := alrRobotPos[iAxis, TManualCmd.e_TeachPos];
					alrCurrentSpeed[iAxis] := aTRobotAxis[iAxis].lrManualSpeed;
				END_FOR

